Fanuc KAREL source: ko00064.KL

-- PROVISIONAL review KL for V1013-1; original PC SHA256 423e0fd4fcb736f2b66a3959d1b53844cb234b2e3040f886e97fb236354ad40f
-- Incomplete behavior may be omitted. Consult companion uncertainty JSON. Do not deploy.
PROGRAM KO00064
%NOLOCKGROUP
BEGIN
  -- UNRESOLVED_PC offsets 5-12; opcodes 9D,23
  -- UNRESOLVED_PC offsets 17-69; opcodes 27,27,49,7E,AD,27,49,7E,AD,22,31,7E,4A
  -- UNRESOLVED_PC offsets 74-78; opcodes 7F
END KO00064
